{attribute addProperty BoxType "EJ9505-0000-0016"}
{attribute addProperty Id "Status_UoAT %I*Status_Uo_D24303661620WcStateAT %I*WcState_F855686C1620InfoDataAT %I*InfoData_192954DE1620"}
{attribute addProperty CRC "4276642424"}
{attribute addProperty SizeInBites "48"}
{attribute addProperty SizeInBytes "6"}
TYPE EJ9505_A1085FEB :
STRUCT
	{attribute addProperty Name "Status_Uo"}
	Status_Uo : Status_Uo_D2430366;
	{attribute addProperty Name "WcState"}
	WcState : WcState_F855686C;
	{attribute addProperty Name "InfoData"}
	InfoData : InfoData_192954DE;
END_STRUCT
END_TYPE

(* stored: Version 1.2.0.0, ProductVersion 3.1.4024.9
   DUT EJ9505_A1085FEB: Id {3104f57e-5e5f-45f6-9d30-8262b9dd34c1} *)
